VAR_GLOBAL
	sOpcUaServerUrl : STRING(MAX_STRING_LENGTH) := 'opc.tcp://localhost:48030';
	sNamespaceUri : STRING(MAX_STRING_LENGTH) := 'http://yourorganisation.org/TcOpcUaSampleServer/';
END_VAR

(* stored: Version 1.1.0.1
   GVL Settings: Id {eb05ed2f-70d2-4892-b1f1-f5dc3e9ac14b} *)
